// This Function is used to avoid division by 0.
// If you integrate these functions in the PLC project, they are called before each division that occurs in the code.
// Implicitly generated code : DO NOT EDIT
FUNCTION CheckDivReal : REAL
VAR_INPUT
	divisor:REAL;
END_VAR

// Implicitly generated code : Only an Implementation suggestion
{noflow}
IF divisor = 0 THEN
	CheckDivReal:=1;
	GVL_TwinCatChecks.CheckDiv_REAL_DivBy0 := GVL_TwinCatChecks.CheckDiv_REAL_DivBy0 + 1;
ELSE
	CheckDivReal:=divisor;
END_IF;
{flow}

END_FUNCTION

(* stored: Version 1.1.0.1, ProductVersion 3.1.4024.10
   POU CheckDivReal: Id {5c7399aa-2e9a-4177-883d-f5eb0a0ffed1}, SpecialFunc CheckDivReal32 *)
